{attribute addProperty BoxType "EK1122-0000-0018"}
{attribute addProperty Id "Beckhoff_ER8xxxsub_EK1100EK1100_179A0949162A_0001_ER8309_1022_0018ER8309_4876315539449.25"}
{attribute addProperty CRC "96784593"}
{attribute addProperty SizeInBites "410"}
{attribute addProperty SizeInBytes "51.25"}
TYPE Beckhoff_ER8xxxEK1122_05C4D0D1 EXTENDS EK1122_179A0949 :
STRUCT
	{attribute addProperty Name "Beckhoff_ER8xxxsub_EK1100"}
	Beckhoff_ER8xxxsub_EK1100 : EK1100_179A0949;
	{attribute addProperty Name "A_0001_ER8309_1022_0018"}
	A_0001_ER8309_1022_0018 : ER8309_48763155;
END_STRUCT
END_TYPE

(* stored: Version 1.2.0.0, ProductVersion 3.1.4024.9
   DUT Beckhoff_ER8xxxEK1122_05C4D0D1: Id {217ba566-9e84-45ce-956d-4a02eb923db7} *)
